# EPICS substitutions: SKFMB350/SKFMB350-IOC-01App/Db/status.substitutions
file interlocks.template {

pattern {P, SNAME, FIELD, ZNAM, ONAM}
{"\$(P)", "OK", "B0", "NOT OK", "OK"}
{"\$(P)", "UP_TO_SPEED", "B1", "YES", "NO"}
{"\$(P)", "RUN", "B2", "YES", "NO"}
{"\$(P)", "SHUTDOWN", "B3", "YES", "NO"}
{"\$(P)", "LEVITATION_COMPLETE", "B4", "YES", "NO"}
{"\$(P)", "PHASE_LOCKED", "B5", "YES", "NO"}
{"\$(P)", "DIRECTION", "B6", "Clockwise", "Counter-clockwise"}
{"\$(P)", "AVC_ON", "B7", "YES", "NO"}
}
